TYPE ST_Record :
STRUCT

    nID        : LINT;
    dtTimestamp: DATE_AND_TIME;
    sName      : STRING;
    nSensor1   : LREAL;
    nSensor2   : LREAL;
END_STRUCT
END_TYPE

(* stored: Version 1.1.0.1, ProductVersion 3.1.4022.12
   DUT ST_Record: Id {9397a3ac-c5cf-4c81-a5c1-b5271515bd01} *)
